// Mitsubishi GX Works2 project: 축(인텔리전트 명령)   PLC: Q02/Q02H

PROGRAM MAIN
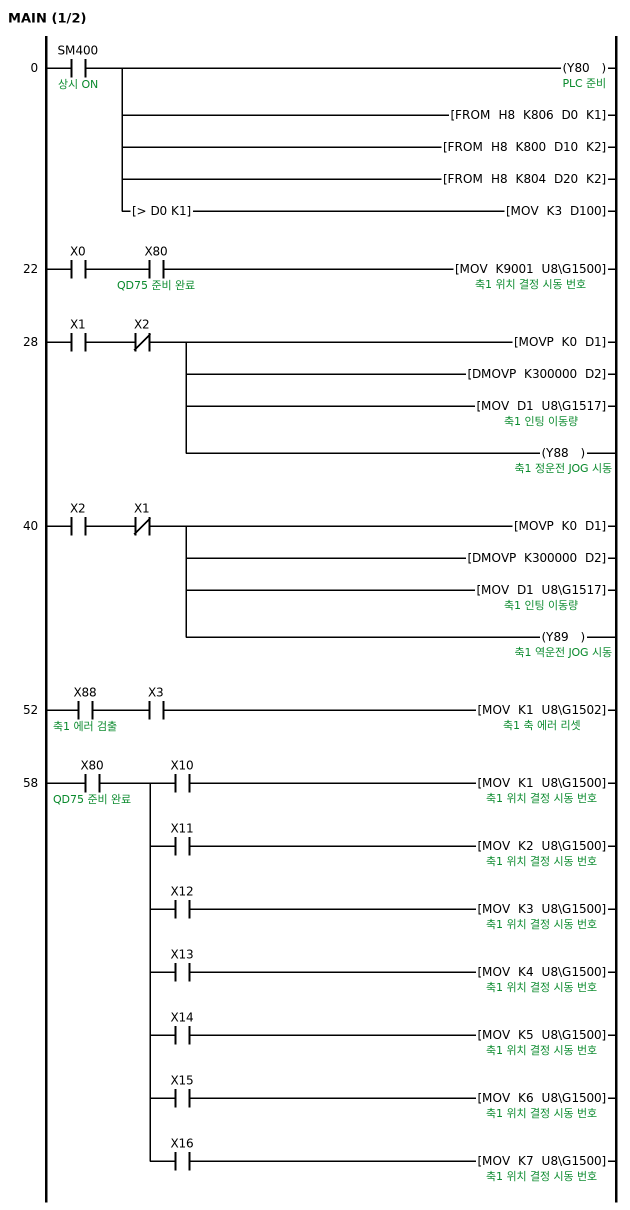
0     LD      SM400  ; 상시 ON
      OUT     Y80  ; PLC 준비
      FROM    H8 K806 D0 K1
      FROM    H8 K800 D10 K2
      FROM    H8 K804 D20 K2
      AND>    D0 K1
      MOV     K3 D100
22    LD      X0
      AND     X80  ; QD75 준비 완료
      MOV     K9001 U8\G1500  ; 축1 위치 결정 시동 번호
28    LD      X1
      ANI     X2
      MOVP    K0 D1
      DMOVP   K300000 D2
      MOV     D1 U8\G1517  ; 축1 인팅 이동량
      OUT     Y88  ; 축1 정운전 JOG 시동
40    LD      X2
      ANI     X1
      MOVP    K0 D1
      DMOVP   K300000 D2
      MOV     D1 U8\G1517
      OUT     Y89  ; 축1 역운전 JOG 시동
52    LD      X88  ; 축1 에러 검출
      AND     X3
      MOV     K1 U8\G1502  ; 축1 축 에러 리셋
58    LD      X80  ; QD75 준비 완료
      MPS
      AND     X10
      MOV     K1 U8\G1500
      MRD
      AND     X11
      MOV     K2 U8\G1500
      MRD
      AND     X12
      MOV     K3 U8\G1500
      MRD
      AND     X13
      MOV     K4 U8\G1500
      MRD
      AND     X14
      MOV     K5 U8\G1500
      MRD
      AND     X15
      MOV     K6 U8\G1500
      MPP
      AND     X16
      MOV     K7 U8\G1500
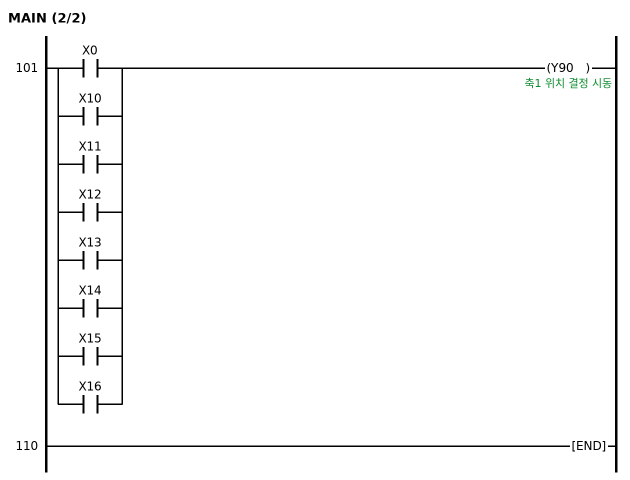
101   LD      X0
      OR      X10
      OR      X11
      OR      X12
      OR      X13
      OR      X14
      OR      X15
      OR      X16
      OUT     Y90  ; 축1 위치 결정 시동
110   END
END_PROGRAM

// device comments not shown above
X81  ; 동기용 플래그
X84  ; 축1 M 코드 ON
X8C  ; 축1 BUSY
X90  ; 축1 시동 완료
X94  ; 축1 위치 결정 완료
Y84  ; 축1 축 정지
Y94  ; 축1 실행 금지 플래그
